FUNCTION FUN_ResetStorageCylinder : BOOL
VAR_INPUT
END_VAR
VAR
END_VAR

END_FUNCTION

(* stored: Version 1.1.0.1, ProductVersion 3.1.4024.13
   POU FUN_ResetStorageCylinder: Id {76d3ec42-64cd-40ee-899e-85d1a5e209a4}, SpecialFunc None *)
